SUBAPPLICATION SubApp_PC_B (* Geraet B (Station 12, 192.168.1.12): schaltet Output_Q1 basierend auf einem lokal ueberwachten OPC-UA-Knoten (AX_SUBSCRIBE_1), der von Geraet A per CLIENT_1_0 remote beschrieben wird - 'SUB style': das Protokoll steckt im MyLib::sys-Composite (logiBUS_QXA_FROM_SUBSCRIBE_OPC), nicht in der Resource des Geraets *)
  (* Standard: 61499-2; Description: Copyright (c) 2026 Meisterschulen am Ostbahnhof This program and the accompanying materials are made available under the terms of the Eclipse Public License 2.0 which is available at https://www.eclipse.org/legal/epl-2.0/ SPDX-License-Identifier: EPL-2.0 *)
  (* Version 1.0, 2026-09-02, Franz Höpfinger, Meisterschulen am Ostbahnhof, initial API and implementation and/or initial documentation *)
  PACKAGE Training_OPC_UA_SUB;
  IMPORT VV::const::OPC_UA::myOpcUaAddresses::Q1_LOCAL_READ;
  IMPORT logiBUS::io::DQ::logiBUS_DO::Output_Q1;
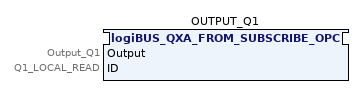
  SUBAPPS
    OUTPUT_Q1 : MyLib::sys::logiBUS_QXA_FROM_SUBSCRIBE_OPC(Output := Output_Q1, ID := Q1_LOCAL_READ);
  END_SUBAPPS
END_SUBAPPLICATION
